FUNCTION_BLOCK MoverSequenceGoHome EXTENDS MoverSequence IMPLEMENTS ZCore.ISequence
VAR
  _step : ZCore.Step(MoverStep.GohomeBegin, MoverStep.GohomeEnd);
  _timer : ZAux.Timer;
END_VAR

IF NOT Busy THEN
  RETURN;
END_IF

IF OnStart(_step) THEN
  ; // init custom sequence variables here ...
END_IF

IF OnStop() THEN
  RETURN; // external stop was triggered
END_IF

IF OnHalt() THEN
  ; // Halting := TRUE; // Uncomment to acknowledge that the sequence is halting
END_IF

REPEAT
  LogStep();

  CASE _step.Index OF
    (* -------------------------------------------------------------------------------------------------------------------------------- *)
    MoverStep.GoHomeBegin:
    (* -------------------------------------------------------------------------------------------------------------------------------- *)
      IF _step.OnEntry()
      THEN
        _timer.WaitAsync(2);
			END_IF
      
      Await(_timer, nextStep:=MoverStep.GoHomeEnd);
      // _step.SetNext(index:=MoverStep.GoHomeEnd);

    (* -------------------------------------------------------------------------------------------------------------------------------- *)
    MoverStep.GoHomeEnd:
    (* -------------------------------------------------------------------------------------------------------------------------------- *)
      SetBusy(FALSE);
  
  ELSE
    Abort('sequence contains unhandled step');
  END_CASE
UNTIL _step.IsNotRepeatable() OR_ELSE NOT Busy END_REPEAT

END_FUNCTION_BLOCK

(* stored: Version 1.1.0.1
   POU MoverSequenceGoHome: Id {1080645a-6ad2-40eb-afd5-6c9bda07b22a}, SpecialFunc None *)
